// TIA Portal V19 export
TYPE "MES_Err_&_Msg"
// stored: Access Published
   STRUCT
      Presence : Bool;
      Code : DInt;
      Description : String;
      Msg : "MES_Msg";   // Messaggio che ha causato errore
   END_STRUCT;
END_TYPE
